TYPE ST_CONTROL_SIGNALS_SETTINGS EXTENDS ST_BASE_SETTINGS:
STRUCT
	// All of them are under VAR_STAT
END_STRUCT
END_TYPE

(* stored: Version 1.1.0.1, ProductVersion 3.1.4026.18
   DUT ST_CONTROL_SIGNALS_SETTINGS: Id {371ff20b-7364-43aa-99e9-be71aa561f4b} *)
